TYPE ST120_PnpHorPos_e : ST110_PnpHorPos_e;
END_TYPE

(* stored: Version 1.1.0.1, ProductVersion 3.1.4024.6
   DUT ST120_PnpHorPos_e: Id {7a5cb5d1-2048-4d8c-94aa-29d61dcfc1bd} *)
